LIN {X 0,Y 82.643,Z 604.93,A -85,B 0,C 180,E1 -30252.083,E2 -30252.083} C_VEL
LIN {X 0,Y 72.722,Z 611.136,A -85,B 0,C 180,E1 -30254.919,E2 -30254.919} C_VEL
LIN {X 0,Y 59.862,Z 617.698,A -85,B 0,C 180,E1 -30260.105,E2 -30260.105} C_VEL
LIN {X 0,Y 47.806,Z 622.616,A -85,B 0,C 180,E1 -30268.131,E2 -30268.131} C_VEL
LIN {X 0,Y 37.125,Z 626.033,A -85,B 0,C 180,E1 -30280.801,E2 -30280.801} C_VEL
LIN {X 0,Y 29.496,Z 628.053,A -85,B 0,C 180,E1 -30301.56,E2 -30301.56} C_VEL
LIN {X 0,Y 27.007,Z 628.715,A -85,B 0,C 180,E1 -30330.019,E2 -30330.019} C_VEL
LIN {X 0,Y 29.504,Z 628.015,A -85,B 0,C 180,E1 -30358.47,E2 -30358.47} C_VEL
LIN {X 0,Y 37.139,Z 625.963,A -85,B 0,C 180,E1 -30379.216,E2 -30379.216} C_VEL
LIN {X 0,Y 42.266,Z 624.419,A -85,B 0,C 180,E1 -30386.264,E2 -30386.264} C_VEL
LIN {X 0,Y 42.738,Z 623.889,A -85,B 0,C 180,E1 -30390.441,E2 -30390.441} C_VEL
LIN {X 0,Y 50.304,Z 621.121,A -85,B 0,C 180,E1 -30444.781,E2 -30444.781} C_VEL
LIN {X 0,Y 48.14,Z 622.155,A -85,B 0,C 180,E1 -30448.822,E2 -30448.822} C_VEL
LIN {X 0,Y 37.433,Z 625.577,A -85,B 0,C 180,E1 -30461.304,E2 -30461.304} C_VEL
LIN {X 0,Y 29.694,Z 627.605,A -85,B 0,C 180,E1 -30481.728,E2 -30481.728} C_VEL
LIN {X 0,Y 27.068,Z 628.291,A -85,B 0,C 180,E1 -30509.981,E2 -30509.981} C_VEL
LIN {X 0,Y 29.68,Z 627.647,A -85,B 0,C 180,E1 -30538.248,E2 -30538.248} C_VEL
LIN {X 0,Y 37.394,Z 625.655,A -85,B 0,C 180,E1 -30558.724,E2 -30558.724} C_VEL
LIN {X 0,Y 48.094,Z 622.267,A -85,B 0,C 180,E1 -30571.233,E2 -30571.233} C_VEL
LIN {X 0,Y 60.112,Z 617.382,A -85,B 0,C 180,E1 -30579.254,E2 -30579.254} C_VEL
LIN {X 0,Y 69.648,Z 612.645,A -85,B 0,C 180,E1 -30583.433,E2 -30583.433} C_VEL
LIN {X 0,Y 81.147,Z 605.78,A -85,B 0,C 180,E1 -30586.963,E2 -30586.963} C_VEL
LIN {X 0,Y 92.857,Z 597.249,A -85,B 0,C 180,E1 -30589.677,E2 -30589.677} C_VEL
LIN {X 0,Y 94.762,Z 595.442,A -85,B 0,C 180,E1 -30591.469,E2 -30591.469} C_VEL
LIN {X 0,Y 95.517,Z 594.314,A -85,B 0,C 180,E1 -30594.668,E2 -30594.668} C_VEL
LIN {X 0,Y 95.313,Z 594.361,A -85,B 0,C 180,E1 -30595.955,E2 -30595.955} C_VEL
LIN {X 0,Y 93.639,Z 595.628,A -85,B 0,C 180,E1 -30597.896,E2 -30597.896} C_VEL
LIN {X 0,Y 91.325,Z 597.396,A -85,B 0,C 180,E1 -30600.373,E2 -30600.373} C_VEL
LIN {X 0,Y 90.993,Z 597.675,A -85,B 0,C 180,E1 -30601.349,E2 -30601.349} C_VEL
LIN {X 0,Y 90.749,Z 598.084,A -85,B 0,C 180,E1 -30604.441,E2 -30604.441} C_VEL
LIN {X 0,Y 89.205,Z 599.436,A -85,B 0,C 180,E1 -30605.934,E2 -30605.934} C_VEL
LIN {X 0,Y 78.03,Z 607.095,A -85,B 0,C 180,E1 -30607.851,E2 -30607.851} C_VEL
LIN {X 0,Y 67.833,Z 612.881,A -85,B 0,C 180,E1 -30610.221,E2 -30610.221} C_VEL
LIN {X 0,Y 57.796,Z 617.644,A -85,B 0,C 180,E1 -30613.434,E2 -30613.434} C_VEL
LIN {X 0,Y 44.882,Z 622.562,A -85,B 0,C 180,E1 -30620.063,E2 -30620.063} C_VEL
LIN {X 0,Y 32.907,Z 625.978,A -85,B 0,C 180,E1 -30631.351,E2 -30631.351} C_VEL
LIN {X 0,Y 23.475,Z 627.997,A -85,B 0,C 180,E1 -30653.246,E2 -30653.246} C_VEL
LIN {X 0,Y 19.902,Z 628.659,A -85,B 0,C 180,E1 -30690.026,E2 -30690.026} C_VEL
LIN {X 0,Y 23.485,Z 627.959,A -85,B 0,C 180,E1 -30726.789,E2 -30726.789} C_VEL
LIN {X 0,Y 32.924,Z 625.907,A -85,B 0,C 180,E1 -30748.661,E2 -30748.661} C_VEL
LIN {X 0,Y 34.268,Z 625.563,A -85,B 0,C 180,E1 -30750.372,E2 -30750.372} C_VEL
LIN {X 0,Y 34.452,Z 625.199,A -85,B 0,C 180,E1 -30755.923,E2 -30755.923} C_VEL
LIN {X 0,Y 40.626,Z 623.5,A -85,B 0,C 180,E1 -30802.343,E2 -30802.343} C_VEL
LIN {X 0,Y 38.971,Z 624.102,A -85,B 0,C 180,E1 -30805.589,E2 -30805.589} C_VEL
LIN {X 0,Y 27.963,Z 626.816,A -85,B 0,C 180,E1 -30821.034,E2 -30821.034} C_VEL
LIN {X 0,Y 20.814,Z 628.171,A -85,B 0,C 180,E1 -30850.24,E2 -30850.24} C_VEL
LIN {X 0,Y 19.976,Z 628.346,A -85,B 0,C 180,E1 -30869.975,E2 -30869.975} C_VEL
LIN {X 0,Y 23.658,Z 627.702,A -85,B 0,C 180,E1 -30906.424,E2 -30906.424} C_VEL
LIN {X 0,Y 33.122,Z 625.71,A -85,B 0,C 180,E1 -30928.046,E2 -30928.046} C_VEL
LIN {X 0,Y 45.094,Z 622.322,A -85,B 0,C 180,E1 -30939.215,E2 -30939.215} C_VEL
LIN {X 0,Y 57.967,Z 617.436,A -85,B 0,C 180,E1 -30945.876,E2 -30945.876} C_VEL
LIN {X 0,Y 67.957,Z 612.698,A -85,B 0,C 180,E1 -30949.212,E2 -30949.212} C_VEL
LIN {X 0,Y 79.84,Z 605.831,A -85,B 0,C 180,E1 -30951.96,E2 -30951.96} C_VEL
LIN {X 0,Y 88.405,Z 599.961,A -85,B 0,C 180,E1 -30953.518,E2 -30953.518} C_VEL
LIN {X 0,Y 90.003,Z 598.558,A -85,B 0,C 180,E1 -30955.521,E2 -30955.521} C_VEL
LIN {X 0,Y 91.183,Z 597.496,A -85,B 0,C 180,E1 -30960,E2 -30960} C_VEL
LIN {X 0,Y 90.993,Z 597.675,A -85,B 0,C 180,E1 -30961.349,E2 -30961.349} C_VEL
LIN {X 0,Y 90.29,Z 598.276,A -85,B 0,C 180,E1 -30962.41,E2 -30962.41} C_VEL
LIN {X 0,Y 88.524,Z 599.671,A -85,B 0,C 180,E1 -30963.264,E2 -30963.264} C_VEL
LIN {X 0,Y 85.412,Z 601.898,A -85,B 0,C 180,E1 -30963.71,E2 -30963.71} C_VEL
LIN {X 0,Y 75.46,Z 608.187,A -85,B 0,C 180,E1 -30963.013,E2 -30963.013} C_VEL
LIN {X 0,Y 73.377,Z 609.362,A -85,B 0,C 180,E1 -30963.175,E2 -30963.175} C_VEL
LIN {X 0,Y 60.012,Z 616.131,A -85,B 0,C 180,E1 -30965.573,E2 -30965.573} C_VEL
LIN {X 0,Y 49.721,Z 620.244,A -85,B 0,C 180,E1 -30968.407,E2 -30968.407} C_VEL
LIN {X 0,Y 36.312,Z 624.395,A -85,B 0,C 180,E1 -30974.652,E2 -30974.652} C_VEL
LIN {X 0,Y 23.699,Z 627.103,A -85,B 0,C 180,E1 -30987.216,E2 -30987.216} C_VEL
LIN {X 0,Y 14.196,Z 628.442,A -85,B 0,C 180,E1 -31020.368,E2 -31020.368} C_VEL
LIN {X 0,Y 12.79,Z 628.603,A -85,B 0,C 180,E1 -31050.04,E2 -31050.04} C_VEL
LIN {X 0,Y 18.286,Z 627.903,A -85,B 0,C 180,E1 -31100.276,E2 -31100.276} C_VEL
LIN {X 0,Y 25.693,Z 626.674,A -85,B 0,C 180,E1 -31115.746,E2 -31115.746} C_VEL
LIN {X 0,Y 26.7,Z 626.275,A -85,B 0,C 180,E1 -31124.74,E2 -31124.74} C_VEL
LIN {X 0,Y 29.533,Z 625.601,A -85,B 0,C 180,E1 -31153.768,E2 -31153.768} C_VEL
LIN {X 0,Y 29.994,Z 625.689,A -85,B 0,C 180,E1 -31160.36,E2 -31160.36} C_VEL
LIN {X 0,Y 18.432,Z 627.717,A -85,B 0,C 180,E1 -31180.265,E2 -31180.265} C_VEL
LIN {X 0,Y 12.873,Z 628.402,A -85,B 0,C 180,E1 -31229.96,E2 -31229.96} C_VEL
LIN {X 0,Y 18.413,Z 627.758,A -85,B 0,C 180,E1 -31279.72,E2 -31279.72} C_VEL
LIN {X 0,Y 29.963,Z 625.766,A -85,B 0,C 180,E1 -31299.705,E2 -31299.705} C_VEL
LIN {X 0,Y 43.077,Z 622.376,A -85,B 0,C 180,E1 -31308.149,E2 -31308.149} C_VEL
LIN {X 0,Y 56.652,Z 617.49,A -85,B 0,C 180,E1 -31312.873,E2 -31312.873} C_VEL
LIN {X 0,Y 66.991,Z 612.751,A -85,B 0,C 180,E1 -31315.206,E2 -31315.206} C_VEL
LIN {X 0,Y 79.158,Z 605.882,A -85,B 0,C 180,E1 -31317.081,E2 -31317.081} C_VEL
LIN {X 0,Y 84.393,Z 602.452,A -85,B 0,C 180,E1 -31317.724,E2 -31317.724} C_VEL
LIN {X 0,Y 85.269,Z 601.82,A -85,B 0,C 180,E1 -31320,E2 -31320} C_VEL
LIN {X 0,Y 84.367,Z 602.494,A -85,B 0,C 180,E1 -31321.781,E2 -31321.781} C_VEL
LIN {X 0,Y 73.377,Z 609.362,A -85,B 0,C 180,E1 -31323.175,E2 -31323.175} C_VEL
LIN {X 0,Y 67.39,Z 612.588,A -85,B 0,C 180,E1 -31323.575,E2 -31323.575} C_VEL
LIN {X 0,Y 57.057,Z 617.25,A -85,B 0,C 180,E1 -31322.705,E2 -31322.705} C_VEL
LIN {X 0,Y 48.575,Z 620.423,A -85,B 0,C 180,E1 -31321.643,E2 -31321.643} C_VEL
LIN {X 0,Y 42.094,Z 622.478,A -85,B 0,C 180,E1 -31321.649,E2 -31321.649} C_VEL
LIN {X 0,Y 39.929,Z 623.058,A -85,B 0,C 180,E1 -31322.03,E2 -31322.03} C_VEL
LIN {X 0,Y 28.248,Z 625.868,A -85,B 0,C 180,E1 -31325.819,E2 -31325.819} C_VEL
LIN {X 0,Y 14.761,Z 627.886,A -85,B 0,C 180,E1 -31337.898,E2 -31337.898} C_VEL
LIN {X 0,Y 8.758,Z 628.386,A -85,B 0,C 180,E1 -31356.731,E2 -31356.731} C_VEL
LIN {X 0,Y 5.691,Z 628.548,A -85,B 0,C 180,E1 -31410.089,E2 -31410.089} C_VEL
LIN {X 0,Y 8.772,Z 628.366,A -85,B 0,C 180,E1 -31463.339,E2 -31463.339} C_VEL
LIN {X 0,Y 18.795,Z 627.356,A -85,B 0,C 180,E1 -31487.596,E2 -31487.596} C_VEL
LIN {X 0,Y 19.751,Z 627.194,A -85,B 0,C 180,E1 -31493.926,E2 -31493.926} C_VEL
LIN {X 0,Y 21.023,Z 626.988,A -85,B 0,C 180,E1 -31509.027,E2 -31509.027} C_VEL
LIN {X 0,Y 19.302,Z 627.239,A -85,B 0,C 180,E1 -31512.992,E2 -31512.992} C_VEL
LIN {X 0,Y 8.844,Z 628.283,A -85,B 0,C 180,E1 -31537.286,E2 -31537.286} C_VEL
LIN {X 0,Y 5.763,Z 628.458,A -85,B 0,C 180,E1 -31589.912,E2 -31589.912} C_VEL
LIN {X 0,Y 14.839,Z 627.814,A -85,B 0,C 180,E1 -31661.195,E2 -31661.195} C_VEL
LIN {X 0,Y 28.291,Z 625.821,A -85,B 0,C 180,E1 -31673.39,E2 -31673.39} C_VEL
LIN {X 0,Y 42.193,Z 622.431,A -85,B 0,C 180,E1 -31677.698,E2 -31677.698} C_VEL
LIN {X 0,Y 49.194,Z 620.182,A -85,B 0,C 180,E1 -31679.012,E2 -31679.012} C_VEL
LIN {X 0,Y 49.976,Z 619.912,A -85,B 0,C 180,E1 -31679.999,E2 -31679.999} C_VEL
LIN {X 0,Y 39.929,Z 623.058,A -85,B 0,C 180,E1 -31682.03,E2 -31682.03} C_VEL
LIN {X 0,Y 39.929,Z 623.058,A -85,B 0,C 180,E1 -31682.03,E2 -31682.03}

QRS_NEXT_CUT()

QRS_NEXT()
QRS_HOME()

END
